(*
SPDX-FileCopyrightText: © 2026 Oleksandr Tiutyk <trofimich@gmail.com>
SPDX-License-Identifier: MIT
License: https://opensource.org/license/mit
*)

(*!
<summary>Provides generic-value insertion, replacement, removal and in-place reordering.</summary>
<description>
Successful insertion transfers disposal responsibility for owned payload; borrowed payload must remain alive
while stored. The caller-side descriptor copy is not reset and must not be released again after transfer.
Independent owning aliases and overlapping owned allocations are unsupported. Get and FindSingle do not
transfer ownership back. Removal releases owned payload. Validators are borrowed. Sort and Swap change entry
order without changing collection length or payload ownership. Same-allocation replacement preserves
collection ownership; aliases must have compatible disposal semantics.
</description>
*)

INTERFACE IList EXTENDS IReadOnlyList

(*!
<summary>Copies a value and appends the owned descriptor.</summary>
<description>
Borrows the original during the call. isObject = TRUE requires a live Object FB instance implementing
ICloneable; other data is copied as bytes without recursively cloning references. A prepared copy is released
if insertion fails before acceptance; exceptions propagate. Engine-managed exception objects are unsupported.
index is meaningful only on success.
The original exception is captured before prepared-copy cleanup, so nested cleanup handling cannot replace
its payload. Terminal OOM takes precedence; capture failure still attempts prepared-copy disposal.
</description>
*)
METHOD AppendCopy : IList
VAR_INPUT
	value : ANY;
	isObject : BOOL := FALSE;
END_VAR
VAR_OUTPUT
	index : TOF_Core.DINT_INDEX;
END_VAR
END_METHOD

(*!
<summary>Appends a descriptor to the list.</summary>
<description>
Successful insertion transfers disposal responsibility for owned payload; borrowed payload must remain alive
while stored. The caller-side descriptor copy is not reset and must not be released again after transfer.
Independent owning aliases and overlapping owned allocations are unsupported. Delegates to InsertGeneric;
index is meaningful only on success.
</description>
*)
METHOD AppendGeneric : IList
VAR_INPUT
	value : TOF_Core.GENERIC_VALUE;
END_VAR
VAR_OUTPUT
	index : TOF_Core.DINT_INDEX;
END_VAR
END_METHOD

(*!
<summary>Removes all entries and releases dynamic backing storage.</summary>
<description>
Owned payload is released best effort through GENERIC_VALUE.Release; borrowed storage is not freed. Static
capacity and the borrowed validator are retained. Dynamic capacity becomes zero. Returns this collection and
invalidates positions and views. Cleanup callbacks must not reenter mutation.
</description>
*)
METHOD Clear : IList
END_METHOD

(*!
<summary>Reports whether storage can grow dynamically.</summary>
<description>
Static capacity zero selects dynamic storage. Dynamic collections can still fail to allocate.
</description>
*)
{attribute 'monitoring' := 'call'}
PROPERTY Dynamic : BOOL
GET
END_GET
END_PROPERTY

(*!
<summary>Copies a value and inserts it at the requested position.</summary>
<description>
Borrows the original during the call. isObject = TRUE requires a live Object FB instance implementing
ICloneable; other data is copied as bytes without recursively cloning references. A prepared copy is released
if insertion fails before acceptance; exceptions propagate. Engine-managed exception objects are unsupported.
The position may range from zero through Length inclusive.
The original exception is captured before prepared-copy cleanup, so nested cleanup handling cannot replace
its payload. Terminal OOM takes precedence; capture failure still attempts prepared-copy disposal.
</description>
*)
METHOD InsertCopy : IList
VAR_INPUT
	index : TOF_Core.DINT_INDEX;
	value : ANY;
	isObject : BOOL := FALSE;
END_VAR
END_METHOD

(*!
<summary>Inserts a descriptor and shifts subsequent entries to the right.</summary>
<description>
Successful insertion transfers disposal responsibility for owned payload; borrowed payload must remain alive
while stored. The caller-side descriptor copy is not reset and must not be released again after transfer.
Independent owning aliases and overlapping owned allocations are unsupported. index may range from zero
through Length inclusive. Invalid indices and full static storage raise exceptions. Validation precedes
insertion. Dynamic growth rejects nonpositive increments and unrepresentable capacity or allocation sizes
before insertion.
</description>
*)
METHOD InsertGeneric : IList
VAR_INPUT
	index : TOF_Core.DINT_INDEX;
	value : TOF_Core.GENERIC_VALUE;	
END_VAR
END_METHOD

(*!
<summary>Removes an existing list entry and compacts subsequent entries.</summary>
<description>
Invalid indices raise an exception. Owned payload is released best effort through GENERIC_VALUE.Release;
borrowed payload is not freed. Returns this list. Positions and descriptor references may change; cleanup
callbacks must not reenter mutation.
</description>
*)
METHOD RemoveAt : IList
VAR_INPUT
	index : TOF_Core.DINT_INDEX;
END_VAR
END_METHOD

(*!
<summary>Removes the first list entry equal to a borrowed query.</summary>
<description>
Uses default GENERIC_VALUE equality; isObject = TRUE requires a live Object FB instance. Reports removed on a
successful match and returns this list. Owned stored payload is released; the query is not adopted or
separately released. Equality exceptions propagate.
</description>
*)
METHOD RemoveFirst : IList
VAR_INPUT
	value : ANY;
	isObject : BOOL := FALSE;
END_VAR
VAR_OUTPUT
	removed : BOOL;
END_VAR
END_METHOD

(*!
<summary>Removes predicate matches while traversing from the end.</summary>
<description>
skip counts matches from the end. A null predicate or maxRemoved = 0 performs no removal. Removes at most
maxRemoved matching entries after skipping the requested matches. Stops immediately after reaching the limit,
without invoking the predicate for remaining entries. Predicate exceptions propagate after any completed
removals, without rollback. removedCount counts completed removals. Callbacks must not mutate the traversed
collection.
</description>
*)
METHOD RemoveMatched : IList
VAR_INPUT
	predicate : TOF_Core.IPredicate;
	skip : UDINT := 0;
	maxRemoved : UDINT := TOF_Core.UnsignedInt32.MAX_VALUE;
END_VAR
VAR_OUTPUT
	removedCount : DINT;
END_VAR
END_METHOD

(*!
<summary>Copies a value and stores it through SetGeneric.</summary>
<description>
Borrows the original during the call. isObject = TRUE requires a live Object FB instance implementing
ICloneable; other data is copied as bytes without recursively cloning references. A prepared copy is released
if insertion fails before acceptance; exceptions propagate. Engine-managed exception objects are unsupported.
Any index output is meaningful only on success.
The original exception is captured before prepared-copy cleanup, so nested cleanup handling cannot replace
its payload. Terminal OOM takes precedence; capture failure still attempts prepared-copy disposal.
</description>
*)
METHOD SetCopy : IList
VAR_INPUT
	index : TOF_Core.DINT_INDEX;
	value : ANY;
	isObject : BOOL := FALSE;
END_VAR
END_METHOD

(*!
<summary>Replaces the descriptor at an existing list position.</summary>
<description>
Successful replacement transfers disposal responsibility for owned payload; borrowed payload must remain alive
while stored. The caller-side descriptor copy is not reset and must not be released again after transfer.
Invalid indices and rejected validation raise exceptions before replacement. Reusing the same allocation
preserves existing ownership or accepts incoming ownership without releasing that allocation. Aliases must
have compatible disposal semantics; independently owned aliases and overlapping owned ranges are unsupported.
A different displaced allocation is released best effort after installing the new descriptor. Cleanup
callbacks must not reenter collection mutation.
</description>
*)
METHOD SetGeneric : IList
VAR_INPUT
	index : TOF_Core.DINT_INDEX;
	value : TOF_Core.GENERIC_VALUE;	
END_VAR
END_METHOD

(*!
<summary>Reorders list entries according to a generic-value comparer.</summary>
<description>
An omitted or null comparer selects GENERIC_VALUE.CompareTo. An explicit comparer takes precedence and must
provide a consistent order for the borrowed stored values. The default order follows Core numeric, text,
temporal and OBJECT rules; incompatible pairs raise GenericConversionNotSupportedException and OBJECT needs
IComparable. Empty/single lists return without comparing. Callbacks must not mutate operands or the list.
Comparison failure may leave entries partially reordered; all descriptors and payload ownership are retained.
</description>
*)
//!<param name="comparer">Optional borrowed ordering strategy; zero selects GENERIC_VALUE.CompareTo.</param>
//!<param name="direction">Requested ordering direction.</param>
METHOD Sort : IList
VAR_INPUT
	comparer : TOF_Core.IComparer := 0;
	direction : TOF_Core.SORT_DIRECTION := TOF_Core.SORT_DIRECTION.ASCENDING;
END_VAR
END_METHOD

(*!
<summary>Exchanges two positions without cloning or releasing payload.</summary>
<description>
Returns this list. Different indices must be valid or an exception is raised. Current implementation returns
immediately for equal indices without validating them. Payload ownership is preserved.
</description>
*)
METHOD Swap : IList
VAR_INPUT
	index1 : TOF_Core.DINT_INDEX;
	index2 : TOF_Core.DINT_INDEX;
END_VAR
END_METHOD

(*!
<summary>Exposes the configured value validator.</summary>
<description>
Borrowed optional reference fixed at initialization. Zero means no validator. The collection does not own or
release it.
</description>
*)
{attribute 'monitoring' := 'call'}
PROPERTY ValueValidator : TOF_Core.IGenericValueValidator
GET
END_GET
END_PROPERTY

END_INTERFACE

(* stored: Version 1.1.0.1
   Itf IList: Id {9c3b1d1d-e3a1-4bce-bd52-5e0052f367c5}
   Method AppendCopy: Id {ac3e836f-588d-4e01-b78d-500901973fe6}
   Method AppendGeneric: Id {1c7613bb-2dbe-4c5d-a556-c22fe102712a}
   Method Clear: Id {ba38f8c3-7bfc-4319-b27d-1f0e4f4a811e}
   Property Dynamic: Id {71fa123f-357a-4471-a15d-77d645a96458}
   Get Get: Id {f7756e60-d4c6-4ce3-b03c-201c59df0dc2}
   Method InsertCopy: Id {5cb4df9f-a6c0-45ea-9622-2c963ebd948e}
   Method InsertGeneric: Id {87183fae-0fce-4e39-9ddd-d90d34c30a32}
   Method RemoveAt: Id {0b8aa929-5f9c-41a5-aea3-f997d9db63e1}
   Method RemoveFirst: Id {aef0ca9c-d714-4a50-863d-5b01a18245b0}
   Method RemoveMatched: Id {a4ece42e-52ea-4d71-9b54-b1ead6bc0e27}
   Method SetCopy: Id {dd495513-6def-416e-84d8-dbee11dfb071}
   Method SetGeneric: Id {561f245e-a04a-4b0f-9829-137533e39c7a}
   Method Sort: Id {b7150648-9792-4f04-bca7-75d5754e5e7c}
   Method Swap: Id {09e0afcd-004e-4129-b911-deb30ed5603c}
   Property ValueValidator: Id {babf4b9a-7c10-43fe-9d22-162263d6bb72}
   Get Get: Id {89d8735a-6fab-4bd5-8618-8f9f7cbd9223} *)
